{attribute 'GeneratedUsingTerminal: EPP1322-0001-0017'}
{attribute addProperty BoxType "EPP1322-0001-0017"}
{attribute addProperty Id "RC10_AB1_EPP1008_0001EPP1008_78E8D3DD12RC10_AB2_EPP1008_0001EPP1008_78E8D3DD12RC10_AB6_EPP1008_0001EPP1008_78E8D3DD12RC10_AB3_EPP1008_0001EPP1008_78E8D3DD12RC10_AB4_EPP1008_0001EPP1008_78E8D3DD12RC10_AB7_EPP1008_0001EPP1008_78E8D3DD12RC10_AB9_EPP1008_0001EPP1008_78E8D3DD12RC10_AB10_EPP1008_0001EPP1008_78E8D3DD12RC10_AB8_EPP1008_0001EPP1008_78E8D3DD12RC10_AB5_EPP1008_0001EPP1008_78E8D3DD12"}
{attribute addProperty CRC "2165179712"}
{attribute addProperty Size "120"}
{attribute addProperty Name "RC10_EPP (EPP1322-0001)"}
TYPE RC10_EPP_EPP1322_0001_810E0540 EXTENDS EPP1322_1FC0878B :
STRUCT
	{attribute addProperty Name "RC10_AB1 (EPP1008-0001)"}
	{attribute addProperty PreviousPort "RC10_EPP (EPP1322-0001) : D"}
	RC10_AB1_EPP1008_0001 : EPP1008_78E8D3DD;
	{attribute addProperty Name "RC10_AB2 (EPP1008-0001)"}
	{attribute addProperty PreviousPort "RC10_AB1 (EPP1008-0001) : B"}
	RC10_AB2_EPP1008_0001 : EPP1008_78E8D3DD;
	{attribute addProperty Name "RC10_AB6 (EPP1008-0001)"}
	{attribute addProperty PreviousPort "RC10_AB2 (EPP1008-0001) : B"}
	RC10_AB6_EPP1008_0001 : EPP1008_78E8D3DD;
	{attribute addProperty Name "RC10_AB3 (EPP1008-0001)"}
	{attribute addProperty PreviousPort "RC10_AB6 (EPP1008-0001) : B"}
	RC10_AB3_EPP1008_0001 : EPP1008_78E8D3DD;
	{attribute addProperty Name "RC10_AB4 (EPP1008-0001)"}
	{attribute addProperty PreviousPort "RC10_AB3 (EPP1008-0001) : B"}
	RC10_AB4_EPP1008_0001 : EPP1008_78E8D3DD;
	{attribute addProperty Name "RC10_AB7 (EPP1008-0001)"}
	{attribute addProperty PreviousPort "RC10_EPP (EPP1322-0001) : B"}
	RC10_AB7_EPP1008_0001 : EPP1008_78E8D3DD;
	{attribute addProperty Name "RC10_AB9 (EPP1008-0001)"}
	{attribute addProperty PreviousPort "RC10_AB7 (EPP1008-0001) : B"}
	RC10_AB9_EPP1008_0001 : EPP1008_78E8D3DD;
	{attribute addProperty Name "RC10_AB10 (EPP1008-0001)"}
	{attribute addProperty PreviousPort "RC10_AB9 (EPP1008-0001) : B"}
	RC10_AB10_EPP1008_0001 : EPP1008_78E8D3DD;
	{attribute addProperty Name "RC10_AB8 (EPP1008-0001)"}
	{attribute addProperty PreviousPort "RC10_AB10 (EPP1008-0001) : B"}
	RC10_AB8_EPP1008_0001 : EPP1008_78E8D3DD;
	{attribute addProperty Name "RC10_AB5 (EPP1008-0001)"}
	{attribute addProperty PreviousPort "RC10_AB8 (EPP1008-0001) : B"}
	RC10_AB5_EPP1008_0001 : EPP1008_78E8D3DD;
END_STRUCT
END_TYPE

(* stored: Version 1.2.0.0, ProductVersion 3.1.4024.11
   DUT RC10_EPP_EPP1322_0001_810E0540: Id {ec844f67-3fd2-0e5c-33a6-6d7d922d99a3} *)
